TYPE ST_VarInfo :
STRUCT
	DataType	: __SYSTEM.TYPE_CLASS;
	Address		: POINTER TO BYTE;
	Size		: T_VarSize;
END_STRUCT
END_TYPE

(* stored: Version 1.1.0.1, ProductVersion 3.1.4024.14
   DUT ST_VarInfo: Id {69333469-f6ee-0f51-11d9-2128960e6c44} *)
